(* CODESYS project CODESYS SIMULATION II.project

Project tree, tasks and I/O mapping:
  Device : CODESYS Control Win V3, 3S - Smart Software Solutions GmbH, order no. 305021, version 3.5.9.10
    application Application
      libraries: Standard, * (System); SysSocket, 3.5.15.0 (System); SysSocket Interfaces, * (System); SysTypes2 Interfaces, * (System)
      task MainTask (cyclic, interval t#20ms, priority 1) calls PLC_PRG
      program PLC_PRG [ST]
      Symbols
  libraries: VisuSymbols, 3.5.8.0 (System)
  text list GlobalTextList
  global variables GVL
  program POU [ST]
*)

// GVL
VAR_GLOBAL
	entradas_plc1: BYTE;
	salidas_plc1: BYTE;
	salidas_plc2: BYTE;
//TCP
	TCP_COMANDOS_VENTOSAS: BYTE;
	TCP_COMANDOS_LEDS: BYTE;
END_VAR

// Device/Application/PLC_PRG
PROGRAM PLC_PRG
VAR
    BP1, BP2, START, STOP, EMERGENCIA : BOOL;
    SISTEMA_ON, START_ANT, LED_TEST : BOOL;
    NEUMATICA_ON, NEUMATICA_OFF : BOOL;
    VENTOSA_OMEGA_ON : BOOL;
    VENTOSA_OMEGA_OFF : BOOL;
    VENTOSA_PALETIZADOR_ON : BOOL;
    VENTOSA_PALETIZADOR_OFF : BOOL;
    LED1, LED2, LED3, LED4 : BOOL;
    LED5, LED6, LED7, LED8 : BOOL;

    TON_LED : TON;
    tSendTimer : TON;
    tNoDataTimer : TON;

    hServer : RTS_IEC_HANDLE := RTS_INVALID_HANDLE;
    hClient : RTS_IEC_HANDLE := RTS_INVALID_HANDLE;

    serverSockAddr : SOCKADDRESS;
    clientSockAddr : SOCKADDRESS;
    addrLen : DINT;

    serverPort : UINT := 8888;

    xServerCreated : BOOL := FALSE;
    xClientConnected : BOOL := FALSE;

    rxBuffer : ARRAY[0..2] OF BYTE;
    txBuffer : ARRAY[0..4] OF BYTE;

    nBytesReceived : DINT;
    nBytesSent : DINT;

    TCP_COMANDOS_VENTOSAS : BYTE := 0;
    TCP_COMANDOS_LEDS : BYTE := 0;

    bPktReceived : BOOL := FALSE;

    fdRead : SOCKET_FD_SET;
    tvTimeout : SOCKET_TIMEVAL;
    diSelectResult : DINT;
    socketResult : DINT;

    SISTEMA_ON_ANT : BOOL := FALSE;
END_VAR


BP1        := (entradas_plc1 AND 16#01) <> 0;
BP2        := (entradas_plc1 AND 16#02) <> 0;
START      := (entradas_plc1 AND 16#04) <> 0;
STOP       := (entradas_plc1 AND 16#08) <> 0;
EMERGENCIA := (entradas_plc1 AND 16#10) <> 0;


// Seguridad y arranque
IF NOT STOP OR NOT EMERGENCIA THEN

    SISTEMA_ON := FALSE;
    START_ANT := FALSE;
    LED_TEST := FALSE;

ELSE

    IF START AND NOT START_ANT THEN
        SISTEMA_ON := TRUE;
        LED_TEST := TRUE;
    END_IF;

    START_ANT := START;

END_IF;


// Test de LEDs durante 1 segundo
TON_LED(IN := LED_TEST, PT := T#1S);

IF TON_LED.Q THEN
    LED_TEST := FALSE;
END_IF;


// Neumática general
IF SISTEMA_ON AND STOP AND EMERGENCIA THEN
    NEUMATICA_ON := TRUE;
    NEUMATICA_OFF := FALSE;
ELSE
    NEUMATICA_ON := FALSE;
    NEUMATICA_OFF := TRUE;
END_IF;


// Ventosas
IF SISTEMA_ON AND STOP AND EMERGENCIA THEN
    VENTOSA_OMEGA_ON := (TCP_COMANDOS_VENTOSAS AND 16#01) <> 0;
    VENTOSA_PALETIZADOR_ON := (TCP_COMANDOS_VENTOSAS AND 16#02) <> 0;
ELSE
    VENTOSA_OMEGA_ON := FALSE;
    VENTOSA_PALETIZADOR_ON := FALSE;
END_IF;

VENTOSA_OMEGA_OFF := NOT VENTOSA_OMEGA_ON;
VENTOSA_PALETIZADOR_OFF := NOT VENTOSA_PALETIZADOR_ON;


// LEDs
IF LED_TEST THEN

    LED1 := TRUE;
    LED2 := TRUE;
    LED3 := TRUE;
    LED4 := TRUE;
    LED5 := TRUE;
    LED6 := TRUE;
    LED7 := TRUE;
    LED8 := TRUE;

ELSE

    LED1 := (TCP_COMANDOS_LEDS AND 16#01) <> 0;
    LED2 := (TCP_COMANDOS_LEDS AND 16#02) <> 0;
    LED3 := (TCP_COMANDOS_LEDS AND 16#04) <> 0;
    LED4 := (TCP_COMANDOS_LEDS AND 16#08) <> 0;
    LED5 := (TCP_COMANDOS_LEDS AND 16#10) <> 0;
    LED6 := (TCP_COMANDOS_LEDS AND 16#20) <> 0;
    LED7 := (TCP_COMANDOS_LEDS AND 16#40) <> 0;
    LED8 := (TCP_COMANDOS_LEDS AND 16#80) <> 0;

END_IF;


// Salidas PLC 1
salidas_plc1 := 0;

IF VENTOSA_OMEGA_ON        THEN salidas_plc1 := salidas_plc1 OR 16#01; END_IF;
IF VENTOSA_OMEGA_OFF       THEN salidas_plc1 := salidas_plc1 OR 16#02; END_IF;
IF VENTOSA_PALETIZADOR_ON  THEN salidas_plc1 := salidas_plc1 OR 16#04; END_IF;
IF VENTOSA_PALETIZADOR_OFF THEN salidas_plc1 := salidas_plc1 OR 16#08; END_IF;

IF LED7 THEN salidas_plc1 := salidas_plc1 OR 16#10; END_IF;
IF LED8 THEN salidas_plc1 := salidas_plc1 OR 16#20; END_IF;
IF LED5 THEN salidas_plc1 := salidas_plc1 OR 16#40; END_IF;
IF LED6 THEN salidas_plc1 := salidas_plc1 OR 16#80; END_IF;


// Salidas PLC 2
salidas_plc2 := 0;

IF LED2 THEN salidas_plc2 := salidas_plc2 OR 16#01; END_IF;
IF LED1 THEN salidas_plc2 := salidas_plc2 OR 16#02; END_IF;
IF LED4 THEN salidas_plc2 := salidas_plc2 OR 16#04; END_IF;
IF LED3 THEN salidas_plc2 := salidas_plc2 OR 16#08; END_IF;

IF NEUMATICA_OFF THEN salidas_plc2 := salidas_plc2 OR 16#10; END_IF;
IF NEUMATICA_ON  THEN salidas_plc2 := salidas_plc2 OR 16#20; END_IF;


// Bit 2.6: STOP / EMERGENCIA activo
IF NOT STOP OR NOT EMERGENCIA THEN
    salidas_plc2 := salidas_plc2 OR 16#40;
END_IF;


// Envío inmediato cuando el sistema pasa de ON a OFF
IF xClientConnected AND (SISTEMA_ON_ANT AND NOT SISTEMA_ON) THEN

    txBuffer[0] := 16#BB;
    txBuffer[1] := salidas_plc1;
    txBuffer[2] := salidas_plc2;
    txBuffer[3] := entradas_plc1;
    txBuffer[4] := 0;

    SysSockSend(
        hClient,
        ADR(txBuffer),
        SIZEOF(txBuffer),
        0,
        0
    );

END_IF;

SISTEMA_ON_ANT := SISTEMA_ON;


// Crear servidor TCP
IF NOT xServerCreated THEN

    hServer := SysSockCreate(
        SOCKET_AF_INET,
        SOCKET_STREAM,
        SOCKET_IPPROTO_TCP,
        ADR(socketResult)
    );

    IF hServer <> 0 AND hServer <> RTS_INVALID_HANDLE THEN

        serverSockAddr.sin_family := SOCKET_AF_INET;
        serverSockAddr.sin_port := SysSockHtons(serverPort);

        SysSockInetAddr(
            '127.0.0.1',
            ADR(serverSockAddr.sin_addr)
        );

        IF SysSockBind(
            hServer,
            ADR(serverSockAddr),
            SIZEOF(serverSockAddr)
        ) = 0 THEN

            IF SysSockListen(hServer, 1) = 0 THEN
                xServerCreated := TRUE;
            END_IF;

        ELSE

            SysSockClose(hServer);
            hServer := RTS_INVALID_HANDLE;
            xServerCreated := FALSE;

        END_IF;

    END_IF;

END_IF;


// Aceptar cliente TCP
IF xServerCreated AND NOT xClientConnected THEN

    fdRead.fd_count := 1;
    fdRead.fd_array[0] := hServer;

    tvTimeout.tv_sec := 0;
    tvTimeout.tv_usec := 0;

    diSelectResult := TO_DINT(
        SysSockSelect(
            0,
            ADR(fdRead),
            0,
            0,
            ADR(tvTimeout),
            0
        )
    );

    IF diSelectResult > 0 THEN

        addrLen := SIZEOF(clientSockAddr);

        hClient := SysSockAccept(
            hServer,
            ADR(clientSockAddr),
            ADR(addrLen),
            0
        );

        IF hClient <> 0 AND hClient <> RTS_INVALID_HANDLE THEN

            xClientConnected := TRUE;
            TCP_COMANDOS_VENTOSAS := 0;
            TCP_COMANDOS_LEDS := 0;
            bPktReceived := FALSE;

        END_IF;

    END_IF;

END_IF;


// Recibir comandos desde TCP
IF xClientConnected THEN

    fdRead.fd_count := 1;
    fdRead.fd_array[0] := hClient;

    tvTimeout.tv_sec := 0;
    tvTimeout.tv_usec := 0;

    diSelectResult := TO_DINT(
        SysSockSelect(
            0,
            ADR(fdRead),
            0,
            0,
            ADR(tvTimeout),
            0
        )
    );

    IF diSelectResult > 0 THEN

        nBytesReceived := SysSockRecv(
            hClient,
            ADR(rxBuffer),
            SIZEOF(rxBuffer),
            0,
            0
        );

        IF nBytesReceived > 0 THEN

            IF nBytesReceived = 3 AND rxBuffer[0] = 16#AA THEN

                TCP_COMANDOS_VENTOSAS := rxBuffer[1];
                TCP_COMANDOS_LEDS := rxBuffer[2];
                bPktReceived := TRUE;

            END_IF;

        ELSE

            SysSockClose(hClient);
            hClient := RTS_INVALID_HANDLE;
            xClientConnected := FALSE;
            TCP_COMANDOS_VENTOSAS := 0;
            TCP_COMANDOS_LEDS := 0;

        END_IF;

    END_IF;

END_IF;


// Envío periódico hacia TCP
IF xClientConnected THEN

    tSendTimer(IN := NOT tSendTimer.Q, PT := T#50MS);

    IF tSendTimer.Q THEN

        txBuffer[0] := 16#BB;
        txBuffer[1] := salidas_plc1;
        txBuffer[2] := salidas_plc2;
        txBuffer[3] := entradas_plc1;

        IF SISTEMA_ON THEN
            txBuffer[4] := 1;
        ELSE
            txBuffer[4] := 0;
        END_IF;

        nBytesSent := SysSockSend(
            hClient,
            ADR(txBuffer),
            SIZEOF(txBuffer),
            0,
            0
        );

        IF nBytesSent <= 0 AND nBytesSent <> -1 THEN

            SysSockClose(hClient);
            hClient := RTS_INVALID_HANDLE;
            xClientConnected := FALSE;
            TCP_COMANDOS_VENTOSAS := 0;
            TCP_COMANDOS_LEDS := 0;

        END_IF;

    END_IF;

ELSE

    tSendTimer(IN := FALSE, PT := T#50MS);

END_IF;


// Cierre por falta de datos
tNoDataTimer(IN := xClientConnected AND NOT bPktReceived, PT := T#30S);

IF tNoDataTimer.Q THEN

    SysSockClose(hClient);
    hClient := RTS_INVALID_HANDLE;
    xClientConnected := FALSE;
    TCP_COMANDOS_VENTOSAS := 0;
    TCP_COMANDOS_LEDS := 0;

END_IF;

bPktReceived := FALSE;

END_PROGRAM

// POU
PROGRAM POU
VAR
END_VAR

END_PROGRAM
